Staubli VAL3: getObjectPos.pgx

public program getObjectPos(num x_nIdx (dimensions=1), point x_pOrigin (dimensions=1), point& x_pObject[] (dimensions=1), num& x_nError[] (dimensions=1))
  local trsf l_TRSF
  local num l_nObjectOffset
  local trsf l_trPoint
begin
  // This program returns the instantaneous position of the object
  // on the conveyor
  //
  // Input param
  //  x_nIdx      : Index of the object in the queue
  //  x_pOrigin   : Static position of the object (has been taught)
  //
  // Output param
  //  x_pObject  : Position of object in conveyor frame
  //  x_nError   : Error code
  //    0 : No error
  //    1 : No ID available
  //
  // Comments
  // getNextID method must have been invoked
  // -------------------------------------------------------
  //
  x_nError=0
  if nNumbOfUser[x_nIdx]!=0
    //
    call getObjectOffset(x_nIdx,l_nObjectOffset,x_nError)
    //
    if x_nError==0
      l_trPoint=position(x_pOrigin,world)
      if bLinear
        l_TRSF={l_nObjectOffset,0,0,0,0,0}
        //*** Compute instantaneous object position
        x_pObject.trsf=fConveyor.trsf*l_TRSF*!fConveyor.trsf*l_trPoint
      else
        l_TRSF={0,0,0,0,0,l_nObjectOffset}
        //*** Compute instantaneous object position
        // NOT TESTED YET
        x_pObject.trsf=fConveyor.trsf*l_TRSF*!fConveyor.trsf*l_trPoint*!l_TRSF
      endIf
    endIf
  else
    x_nError=1
    if cfg:bLog==true
      nErrVal[0]=x_nIdx
      call ut:addNumToString(sConvNum+"(getObjectPos)>>"+sErrMsgList[x_nError],sMsg,"*",nErrVal)
      logMsg(sMsg)
    endIf
  endIf
end
